Universal Robots PolyScope program: d_2.urp

Program d_2 (installation=ext_control directory=/programs createdIn=5.17.3 lastSavedIn=5.17.3 robotSerialNumber=20245501435)
Calibrated DH parameters: a=[0.000154, -0.137004, -0.385524, -0.00002, 0.000092, 0]; d=[0.162441, 211.794786, -230.585024, 18.923638, 0.099786, 0.09951]; alpha=[1.569493, -0.001902, 0.003874, 1.570111, -1.570167, 0]; deltaTheta=[0, -1.242934, 1.056292, 0.186646, 0.000002, 0.000001]
InitVariablesNode
Robot Program (runOnlyOnce=false)
  MoveL speed 250 mm/s, acceleration 1200 mm/s^2 (useActiveTCP=true) feature=Plane_2
    Waypoint Waypoint_3: TCP in base x=392.667 y=743.317 z=82.42 mm, rx=-1.4016 ry=-1.7845 rz=1.1361 rad; joints [-130.623, -8.504, 29.617, -52.433, -61.398, -160.522] deg; TCP offset x=28.21 y=-96.107 z=-99.69 mm, rx=0 ry=0 rz=0 rad; feature pose in base x=343.605 y=747.803 z=100.778 mm, rx=2.6274 ry=0.0101 rz=1.3113 rad
    Waypoint Waypoint_5 (Relative): relativeFromPosition TCP in base x=392.681 y=743.31 z=82.435 mm, rx=-1.4016 ry=-1.7845 rz=1.1361 rad; joints [-130.624, -8.504, 29.617, -52.433, -61.398, -160.523] deg; TCP in base x=460.304 y=219.862 z=133.544 mm, rx=-1.3705 ry=-1.8311 rz=1.1476 rad; joints [-172.426, -47.356, 106.652, -87.535, -100.174, -182.475] deg
